SUBAPPLICATION Bool8_TO_logiBUS_QXA8 (* 8 generische digitale Ausgaenge (Kanal frei waehlbar), gemeinsam getriggert durch 1 CNF-Event, adapter-basiert. Generisch fuer jede 8-Bit-Ausgangsgruppe. Schwester-Baustein zu MyLib::sys::Bool8_TO_logiBUS_QX8 (dort logiBUS_QX statt QXA-Adapter). *)
  (* Standard: 61499-2 *)
  (* Version 1.0, 2026-09-09, Franz Höpfinger, Meisterschulen am Ostbahnhof, Angelegt beim Portieren von Uebung_060 nach test_AX zur Wiederverwendung. *)
  PACKAGE MyLib::sys;
  IMPORT logiBUS::io::DQ::logiBUS_DO;
  IMPORT logiBUS::io::DQ::logiBUS_DO_S;
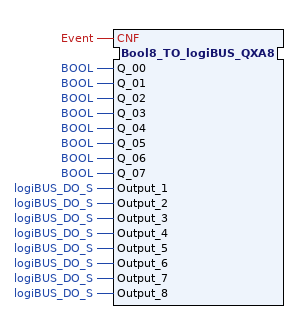
  EVENT_INPUT
    CNF;
  END_EVENT
  VAR_INPUT
    Q_00 : BOOL;
    Q_01 : BOOL;
    Q_02 : BOOL;
    Q_03 : BOOL;
    Q_04 : BOOL;
    Q_05 : BOOL;
    Q_06 : BOOL;
    Q_07 : BOOL;
    Output_1 : logiBUS::io::DQ::logiBUS_DO_S := logiBUS_DO::Invalid; (* Identify the Output Output_Q1..Q8 *)
    Output_2 : logiBUS::io::DQ::logiBUS_DO_S := logiBUS_DO::Invalid; (* Identify the Output Output_Q1..Q8 *)
    Output_3 : logiBUS::io::DQ::logiBUS_DO_S := logiBUS_DO::Invalid; (* Identify the Output Output_Q1..Q8 *)
    Output_4 : logiBUS::io::DQ::logiBUS_DO_S := logiBUS_DO::Invalid; (* Identify the Output Output_Q1..Q8 *)
    Output_5 : logiBUS::io::DQ::logiBUS_DO_S := logiBUS_DO::Invalid; (* Identify the Output Output_Q1..Q8 *)
    Output_6 : logiBUS::io::DQ::logiBUS_DO_S := logiBUS_DO::Invalid; (* Identify the Output Output_Q1..Q8 *)
    Output_7 : logiBUS::io::DQ::logiBUS_DO_S := logiBUS_DO::Invalid; (* Identify the Output Output_Q1..Q8 *)
    Output_8 : logiBUS::io::DQ::logiBUS_DO_S := logiBUS_DO::Invalid; (* Identify the Output Output_Q1..Q8 *)
  END_VAR
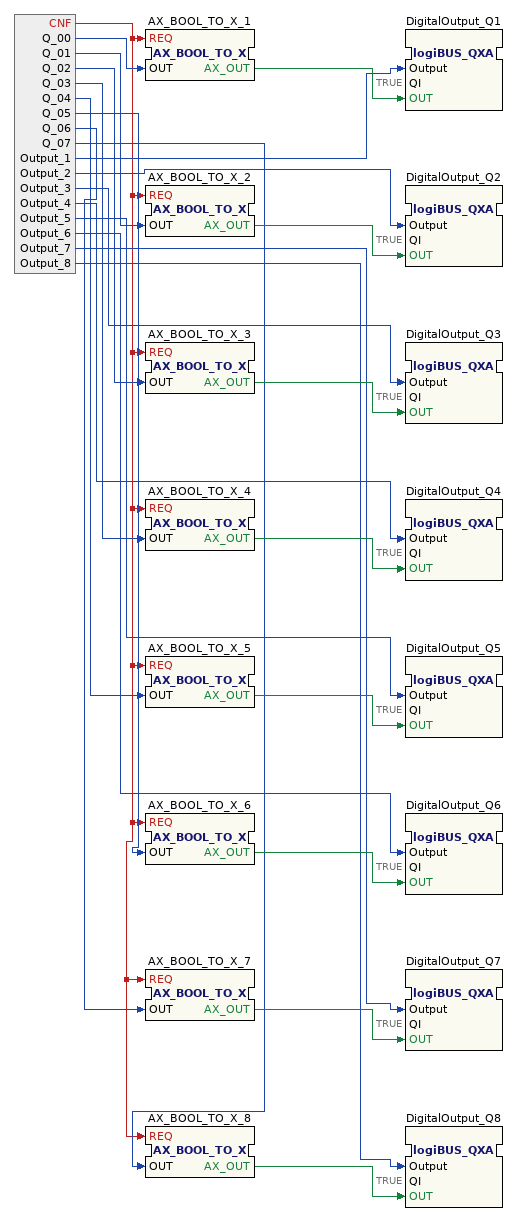
  FBS
    DigitalOutput_Q4 : logiBUS::io::DQ::logiBUS_QXA(QI := TRUE);
    DigitalOutput_Q7 : logiBUS::io::DQ::logiBUS_QXA(QI := TRUE);
    DigitalOutput_Q1 : logiBUS::io::DQ::logiBUS_QXA(QI := TRUE);
    DigitalOutput_Q5 : logiBUS::io::DQ::logiBUS_QXA(QI := TRUE);
    DigitalOutput_Q2 : logiBUS::io::DQ::logiBUS_QXA(QI := TRUE);
    DigitalOutput_Q6 : logiBUS::io::DQ::logiBUS_QXA(QI := TRUE);
    DigitalOutput_Q8 : logiBUS::io::DQ::logiBUS_QXA(QI := TRUE);
    DigitalOutput_Q3 : logiBUS::io::DQ::logiBUS_QXA(QI := TRUE);
    AX_BOOL_TO_X_1 : adapter::conversion::unidirectional::AX_BOOL_TO_X;
    AX_BOOL_TO_X_2 : adapter::conversion::unidirectional::AX_BOOL_TO_X;
    AX_BOOL_TO_X_3 : adapter::conversion::unidirectional::AX_BOOL_TO_X;
    AX_BOOL_TO_X_4 : adapter::conversion::unidirectional::AX_BOOL_TO_X;
    AX_BOOL_TO_X_5 : adapter::conversion::unidirectional::AX_BOOL_TO_X;
    AX_BOOL_TO_X_6 : adapter::conversion::unidirectional::AX_BOOL_TO_X;
    AX_BOOL_TO_X_7 : adapter::conversion::unidirectional::AX_BOOL_TO_X;
    AX_BOOL_TO_X_8 : adapter::conversion::unidirectional::AX_BOOL_TO_X;
  END_FBS
  EVENT_CONNECTIONS
    CNF TO AX_BOOL_TO_X_4.REQ;
    CNF TO AX_BOOL_TO_X_7.REQ;
    CNF TO AX_BOOL_TO_X_1.REQ;
    CNF TO AX_BOOL_TO_X_5.REQ;
    CNF TO AX_BOOL_TO_X_2.REQ;
    CNF TO AX_BOOL_TO_X_6.REQ;
    CNF TO AX_BOOL_TO_X_8.REQ;
    CNF TO AX_BOOL_TO_X_3.REQ;
  END_CONNECTIONS
  DATA_CONNECTIONS
    Q_06 TO AX_BOOL_TO_X_7.OUT;
    Q_00 TO AX_BOOL_TO_X_1.OUT;
    Q_04 TO AX_BOOL_TO_X_5.OUT;
    Q_01 TO AX_BOOL_TO_X_2.OUT;
    Q_05 TO AX_BOOL_TO_X_6.OUT;
    Q_02 TO AX_BOOL_TO_X_3.OUT;
    Q_03 TO AX_BOOL_TO_X_4.OUT;
    Q_07 TO AX_BOOL_TO_X_8.OUT;
    Output_1 TO DigitalOutput_Q1.Output;
    Output_2 TO DigitalOutput_Q2.Output;
    Output_3 TO DigitalOutput_Q3.Output;
    Output_4 TO DigitalOutput_Q4.Output;
    Output_5 TO DigitalOutput_Q5.Output;
    Output_6 TO DigitalOutput_Q6.Output;
    Output_7 TO DigitalOutput_Q7.Output;
    Output_8 TO DigitalOutput_Q8.Output;
  END_CONNECTIONS
  ADAPTER_CONNECTIONS
    AX_BOOL_TO_X_1.AX_OUT TO DigitalOutput_Q1.OUT;
    AX_BOOL_TO_X_2.AX_OUT TO DigitalOutput_Q2.OUT;
    AX_BOOL_TO_X_3.AX_OUT TO DigitalOutput_Q3.OUT;
    AX_BOOL_TO_X_4.AX_OUT TO DigitalOutput_Q4.OUT;
    AX_BOOL_TO_X_5.AX_OUT TO DigitalOutput_Q5.OUT;
    AX_BOOL_TO_X_6.AX_OUT TO DigitalOutput_Q6.OUT;
    AX_BOOL_TO_X_7.AX_OUT TO DigitalOutput_Q7.OUT;
    AX_BOOL_TO_X_8.AX_OUT TO DigitalOutput_Q8.OUT;
  END_CONNECTIONS
END_SUBAPPLICATION
